KUKA KRL data list: Rack_Azul_Cerrar_D.dat

&ACCESS RVO1
&REL 85
&COMMENT CERRAR BANDEJAS PRG
&PARAM EDITMASK = *
&PARAM TEMPLATE = C:\KRC\Roboter\Template\vorgabe
&PARAM DISKPATH = KRC:\R1\Program\MAFELEC
DEFDAT  Rack_Azul_Cerrar_D
;FOLD EXTERNAL DECLARATIONS;%{PE}%MKUKATPBASIS,%CEXT,%VCOMMON,%P
;FOLD GRIPPERTECH EXT
EXT  H50 (INT  :IN,INT  :IN,INT  :IN,GRP_TYP  :IN )
;ENDFOLD (GRIPPERTECH EXT)
;FOLD SPOTTECH EXT
EXT  USERSPOT (S_COMMAND  :IN,SPOT_TYPE  :IN )
;ENDFOLD (SPOTTECH EXT)
;FOLD BASISTECH EXT;%{PE}%MKUKATPBASIS,%CEXT,%VEXT,%P
EXT  BAS (BAS_COMMAND  :IN,REAL  :IN )
DECL INT SUCCESS
;ENDFOLD (BASISTECH EXT)
;FOLD USER EXT;%{E}%MKUKATPUSER,%CEXT,%VEXT,%P
;Make your modifications here

;ENDFOLD (USER EXT)
;ENDFOLD (EXTERNAL DECLARATIONS)
DECL BASIS_SUGG_T LAST_BASIS={POINT1[] "P0                      ",POINT2[] "P0                      ",CP_PARAMS[] "CPDAT0                  ",PTP_PARAMS[] "PDAT0                   ",CONT[] "                        ",CP_VEL[] "1                       ",PTP_VEL[] "100                     ",SYNC_PARAMS[] "SYNCDAT                 ",SPL_NAME[] "S0                      ",A_PARAMS[] "ADAT0                   "}
DECL PDAT PH={VEL 100.000,ACC 100.000,APO_DIST 100.000,APO_MODE #CDIS,GEAR_JERK 50.0000,EXAX_IGN 0}
DECL E6POS XPOS_ESPERA_AREA1={X 112.943756,Y -227.851166,Z 2716.11304,A 36.2463837,B -15.5853510,C 56.0520973,S 3,T 42,E1 0.0,E2 0.0,E3 0.0,E4 0.0,E5 0.0,E6 0.0}
DECL FDAT FPOS_ESPERA_AREA1={TOOL_NO 9,BASE_NO 0,IPO_FRAME #BASE,POINT2[] " ",TQ_STATE FALSE}
DECL LDAT LL={VEL 2.00000,ACC 10.0000,APO_DIST 10.0000,APO_FAC 50.0000,AXIS_VEL 100.000,AXIS_ACC 100.000,ORI_TYP #VAR,CIRC_TYP #BASE,JERK_FAC 50.0000,GEAR_JERK 50.0000,EXAX_IGN 0}
DECL E6POS XPOS_AREA1_LIBRE={X -1304.04749,Y 95.8301,Z 2445.06763,A 84.0317841,B 0.238675669,C -89.1419449,S 6,T 59,E1 0.0,E2 0.0,E3 0.0,E4 0.0,E5 0.0,E6 0.0}
DECL FDAT FPOS_AREA1_LIBRE={TOOL_NO 9,BASE_NO 0,IPO_FRAME #BASE,POINT2[] " ",TQ_STATE FALSE}
DECL E6POS XP111={X 557.799622,Y -753.947571,Z -222.785736,A -88.9974060,B 13.7721291,C 89.1738281,S 6,T 58,E1 0.0,E2 0.0,E3 0.0,E4 0.0,E5 0.0,E6 0.0}
DECL FDAT FP111={TOOL_NO 1,BASE_NO 1,IPO_FRAME #BASE,POINT2[] " ",TQ_STATE FALSE}
DECL E6POS XP10={X 798.959167,Y -279.481934,Z 1381.33276,A 84.0317841,B 0.238675669,C -89.1419449,S 6,T 59,E1 0.0,E2 0.0,E3 0.0,E4 0.0,E5 0.0,E6 0.0}
DECL FDAT FP10={TOOL_NO 1,BASE_NO 2,IPO_FRAME #BASE,POINT2[] " ",TQ_STATE FALSE}
DECL E6POS XP110={X 704.303,Y -173.406952,Z -111.942,A 88.8908,B 0.942831039,C -90.1997757,S 2,T 43,E1 0.0,E2 0.0,E3 0.0,E4 0.0,E5 0.0,E6 0.0}
DECL FDAT FP110={TOOL_NO 2,BASE_NO 2,IPO_FRAME #BASE,POINT2[] " ",TQ_STATE FALSE}
DECL E6POS XP120={X 613.997192,Y -12.6072426,Z 50.9099464,A 86.9020615,B 2.85824347,C -89.1819077,S 2,T 43,E1 0.0,E2 0.0,E3 0.0,E4 0.0,E5 0.0,E6 0.0}
DECL FDAT FP120={TOOL_NO 2,BASE_NO 2,IPO_FRAME #BASE,POINT2[] " ",TQ_STATE FALSE}
DECL E6POS XP_ABRIR10={X -250.533554,Y -43.6507149,Z 2716.11304,A -84.6604385,B 6.50295877,C 57.2217522,S 3,T 42,E1 0.0,E2 0.0,E3 0.0,E4 0.0,E5 0.0,E6 0.0}
DECL FDAT FP_ABRIR10={TOOL_NO 9,BASE_NO 0,IPO_FRAME #BASE,POINT2[] " ",TQ_STATE FALSE}
DECL E6POS XP_AHOME={X -82.6595917,Y 188.465759,Z 3211.91699,A -95.2038803,B -13.5609741,C 10.5279636,S 2,T 43,E1 0.0,E2 0.0,E3 0.0,E4 0.0,E5 0.0,E6 0.0}
DECL FDAT FP_aHOME={TOOL_NO 9,BASE_NO 0,IPO_FRAME #BASE,POINT2[] " ",TQ_STATE FALSE}
DECL E6POS XIni_Cerrar_B1={X 596.412415,Y 736.011475,Z -172.103745,A 87.1854095,B 10.2055225,C -88.9196167,S 2,T 43,E1 0.0,E2 0.0,E3 0.0,E4 0.0,E5 0.0,E6 0.0}
DECL FDAT FIni_Cerrar_B1={TOOL_NO 2,BASE_NO 2,IPO_FRAME #BASE,POINT2[] " ",TQ_STATE FALSE}
DECL E6POS XAux_Cerrar_B1={X 588.737793,Y 569.274475,Z -354.425659,A 86.8103943,B 19.7198429,C -89.4653320,S 2,T 43,E1 0.0,E2 0.0,E3 0.0,E4 0.0,E5 0.0,E6 0.0}
DECL E6POS XFin_Cerrar_B1={X 586.341125,Y 418.554230,Z -648.000366,A 86.3078079,B 27.9656658,C -90.0449677,S 2,T 43,E1 0.0,E2 0.0,E3 0.0,E4 0.0,E5 0.0,E6 0.0}
DECL FDAT FFin_Cerrar_B1={TOOL_NO 2,BASE_NO 2,IPO_FRAME #BASE,POINT2[] "XAux_Cerrar_B1",TQ_STATE FALSE}
DECL E6POS XP0={X 632.645691,Y 303.475861,Z -186.174820,A -88.8950272,B 31.1322117,C 89.5053635,S 6,T 58,E1 0.0,E2 0.0,E3 0.0,E4 0.0,E5 0.0,E6 0.0}
DECL FDAT FP0={TOOL_NO 1,BASE_NO 1,IPO_FRAME #BASE,POINT2[] " ",TQ_STATE FALSE}
DECL E6POS XIni_Cerrar_B2={X 595.075134,Y 739.054,Z 45.4564934,A 87.7715607,B 2.41526031,C -90.0604706,S 2,T 43,E1 0.0,E2 0.0,E3 0.0,E4 0.0,E5 0.0,E6 0.0}
DECL FDAT FIni_Cerrar_B2={TOOL_NO 2,BASE_NO 2,IPO_FRAME #BASE,POINT2[] " ",TQ_STATE FALSE}
DECL E6POS XP1={X 633.606323,Y -740.251,Z -11.7250,A -89.0051498,B 9.17837143,C 89.0890656,S 6,T 58,E1 0.0,E2 0.0,E3 0.0,E4 0.0,E5 0.0,E6 0.0}
DECL FDAT FP1={TOOL_NO 1,BASE_NO 1,IPO_FRAME #BASE,POINT2[] " ",TQ_STATE FALSE}
DECL E6POS XAux_Cerrar_B2={X 587.798340,Y 417.710510,Z -431.910645,A 86.7692,B 24.2213230,C -90.6604462,S 2,T 43,E1 0.0,E2 0.0,E3 0.0,E4 0.0,E5 0.0,E6 0.0}
DECL E6POS XFin_Cerrar_B2={X 589.010254,Y 377.397522,Z -588.953735,A 86.3949585,B 28.6069508,C -90.8338776,S 2,T 43,E1 0.0,E2 0.0,E3 0.0,E4 0.0,E5 0.0,E6 0.0}
DECL FDAT FFin_Cerrar_B2={TOOL_NO 2,BASE_NO 2,IPO_FRAME #BASE,POINT2[] "XAux_Cerrar_B2",TQ_STATE FALSE}
DECL E6POS XP2={X 535.775818,Y 225.276917,Z -536.621948,A -91.0083771,B 14.9493265,C 94.2730637,S 6,T 58,E1 0.0,E2 0.0,E3 0.0,E4 0.0,E5 0.0,E6 0.0}
DECL FDAT FP2={TOOL_NO 1,BASE_NO 1,IPO_FRAME #BASE,POINT2[] " ",TQ_STATE FALSE}
DECL E6POS XP210={X 613.997192,Y -12.6072426,Z 50.9099464,A 86.9020615,B 2.85824347,C -89.1819077,S 2,T 43,E1 0.0,E2 0.0,E3 0.0,E4 0.0,E5 0.0,E6 0.0}
DECL FDAT FP210={TOOL_NO 2,BASE_NO 2,IPO_FRAME #BASE,POINT2[] " ",TQ_STATE FALSE}
DECL E6POS XP220={X 533.749146,Y -27.5535755,Z 294.696930,A 86.9283752,B 2.03337383,C -89.1903,S 2,T 43,E1 0.0,E2 0.0,E3 0.0,E4 0.0,E5 0.0,E6 0.0}
DECL FDAT FP220={TOOL_NO 2,BASE_NO 2,IPO_FRAME #BASE,POINT2[] " ",TQ_STATE FALSE}
DECL E6POS XP3={X 536.241516,Y 225.176605,Z 24.6719704,A -90.9851761,B 14.9447651,C 94.2668762,S 6,T 58,E1 0.0,E2 0.0,E3 0.0,E4 0.0,E5 0.0,E6 0.0}
DECL FDAT FP3={TOOL_NO 1,BASE_NO 1,IPO_FRAME #BASE,POINT2[] " ",TQ_STATE FALSE}
DECL E6POS XIni_Cerrar_B3={X 591.523193,Y 682.249634,Z 258.567474,A 86.9371643,B 3.42378807,C -89.3304749,S 2,T 43,E1 0.0,E2 0.0,E3 0.0,E4 0.0,E5 0.0,E6 0.0}
DECL FDAT FIni_Cerrar_B3={TOOL_NO 2,BASE_NO 2,IPO_FRAME #BASE,POINT2[] " ",TQ_STATE FALSE}
DECL E6POS XP4={X 633.606323,Y -740.251,Z -11.7250,A -89.0051498,B 9.17837143,C 89.0890656,S 6,T 58,E1 0.0,E2 0.0,E3 0.0,E4 0.0,E5 0.0,E6 0.0}
DECL FDAT FP4={TOOL_NO 1,BASE_NO 1,IPO_FRAME #BASE,POINT2[] " ",TQ_STATE FALSE}
DECL E6POS XAux_Cerrar_B3={X 594.214478,Y 611.080200,Z 74.3711472,A 86.8144608,B 12.5334587,C -90.4729614,S 2,T 43,E1 0.0,E2 0.0,E3 0.0,E4 0.0,E5 0.0,E6 0.0}
DECL E6POS XFin_Cerrar_B3={X 594.299866,Y 495.802765,Z -23.1475124,A 86.6915588,B 19.7912579,C -90.9023514,S 2,T 43,E1 0.0,E2 0.0,E3 0.0,E4 0.0,E5 0.0,E6 0.0}
DECL FDAT FFin_Cerrar_B3={TOOL_NO 2,BASE_NO 2,IPO_FRAME #BASE,POINT2[] "XAux_Cerrar_B3",TQ_STATE FALSE}
DECL E6POS XP5={X 535.775818,Y 225.276917,Z -194.099075,A -91.0083771,B 14.9493265,C 94.2730637,S 6,T 58,E1 0.0,E2 0.0,E3 0.0,E4 0.0,E5 0.0,E6 0.0}
DECL FDAT FP5={TOOL_NO 1,BASE_NO 1,IPO_FRAME #BASE,POINT2[] " ",TQ_STATE FALSE}
DECL E6POS XP310={X 533.749146,Y -27.5535755,Z 294.696930,A 86.9283752,B 2.03337383,C -89.1903,S 2,T 43,E1 0.0,E2 0.0,E3 0.0,E4 0.0,E5 0.0,E6 0.0}
DECL FDAT FP310={TOOL_NO 2,BASE_NO 2,IPO_FRAME #BASE,POINT2[] " ",TQ_STATE FALSE}
DECL E6POS XP320={X 530.175537,Y -40.1798019,Z 566.405701,A 86.9635239,B 0.231809333,C -89.0943146,S 2,T 43,E1 0.0,E2 0.0,E3 0.0,E4 0.0,E5 0.0,E6 0.0}
DECL FDAT FP320={TOOL_NO 2,BASE_NO 2,IPO_FRAME #BASE,POINT2[] " ",TQ_STATE FALSE}
DECL E6POS XP310_1={X 593.836731,Y 726.394348,Z 223.429489,A 86.8993149,B 3.44547296,C -89.9683228,S 2,T 43,E1 0.0,E2 0.0,E3 0.0,E4 0.0,E5 0.0,E6 0.0}
DECL FDAT FP310_1={TOOL_NO 2,BASE_NO 2,IPO_FRAME #BASE,POINT2[] " ",TQ_STATE FALSE}
DECL E6POS XP6={X 536.241516,Y 225.176605,Z 24.6719704,A -90.9851761,B 14.9447651,C 94.2668762,S 6,T 58,E1 0.0,E2 0.0,E3 0.0,E4 0.0,E5 0.0,E6 0.0}
DECL FDAT FP6={TOOL_NO 1,BASE_NO 1,IPO_FRAME #BASE,POINT2[] " ",TQ_STATE FALSE}
DECL E6POS XIni_Cerrar_B4={X 582.265930,Y 720.715637,Z 474.957,A 86.9055099,B 6.88711309,C -89.5095520,S 2,T 43,E1 0.0,E2 0.0,E3 0.0,E4 0.0,E5 0.0,E6 0.0}
DECL FDAT FIni_Cerrar_B4={TOOL_NO 2,BASE_NO 2,IPO_FRAME #BASE,POINT2[] " ",TQ_STATE FALSE}
DECL E6POS XP7={X 633.606323,Y -740.251,Z -11.7250,A -89.0051498,B 9.17837143,C 89.0890656,S 6,T 58,E1 0.0,E2 0.0,E3 0.0,E4 0.0,E5 0.0,E6 0.0}
DECL FDAT FP7={TOOL_NO 1,BASE_NO 1,IPO_FRAME #BASE,POINT2[] " ",TQ_STATE FALSE}
DECL E6POS XAux_Cerrar_B4={X 576.527588,Y 424.657928,Z -21.2641106,A 87.9251328,B 24.5308399,C -90.4093552,S 2,T 43,E1 0.0,E2 0.0,E3 0.0,E4 0.0,E5 0.0,E6 0.0}
DECL E6POS XFin_Cerrar_B4={X 576.502,Y 330.746521,Z -306.611084,A 88.2723389,B 22.7116070,C -90.3397293,S 2,T 43,E1 0.0,E2 0.0,E3 0.0,E4 0.0,E5 0.0,E6 0.0}
DECL FDAT FFin_Cerrar_B4={TOOL_NO 2,BASE_NO 2,IPO_FRAME #BASE,POINT2[] "XAux_Cerrar_B4",TQ_STATE FALSE}
DECL E6POS XP8={X 535.775818,Y 225.276917,Z -194.099075,A -91.0083771,B 14.9493265,C 94.2730637,S 6,T 58,E1 0.0,E2 0.0,E3 0.0,E4 0.0,E5 0.0,E6 0.0}
DECL FDAT FP8={TOOL_NO 1,BASE_NO 1,IPO_FRAME #BASE,POINT2[] " ",TQ_STATE FALSE}
DECL E6POS XP410={X 530.175537,Y -40.1798019,Z 566.405701,A 86.9635239,B 0.231809333,C -89.0943146,S 2,T 43,E1 0.0,E2 0.0,E3 0.0,E4 0.0,E5 0.0,E6 0.0}
DECL FDAT FP410={TOOL_NO 2,BASE_NO 2,IPO_FRAME #BASE,POINT2[] " ",TQ_STATE FALSE}
DECL E6POS XP410_1={X 583.801,Y 728.139099,Z 438.754639,A 86.9037552,B 7.08309031,C -89.5218811,S 2,T 43,E1 0.0,E2 0.0,E3 0.0,E4 0.0,E5 0.0,E6 0.0}
DECL FDAT FP410_1={TOOL_NO 2,BASE_NO 2,IPO_FRAME #BASE,POINT2[] " ",TQ_STATE FALSE}
DECL E6POS XP420={X 796.310425,Y -36.4565620,Z 1201.42468,A 84.0344,B 0.236838102,C -89.1263580,S 6,T 59,E1 0.0,E2 0.0,E3 0.0,E4 0.0,E5 0.0,E6 0.0}
DECL FDAT FP420={TOOL_NO 2,BASE_NO 2,IPO_FRAME #BASE,POINT2[] " ",TQ_STATE FALSE}
DECL E6POS XP9={X 536.241516,Y 225.176605,Z 24.6719704,A -90.9851761,B 14.9447651,C 94.2668762,S 6,T 58,E1 0.0,E2 0.0,E3 0.0,E4 0.0,E5 0.0,E6 0.0}
DECL FDAT FP9={TOOL_NO 1,BASE_NO 1,IPO_FRAME #BASE,POINT2[] " ",TQ_STATE FALSE}
DECL E6POS XIni_Cerrar_B5={X 547.158386,Y 717.412231,Z 958.713684,A 91.7971573,B 9.40811539,C -90.5130844,S 6,T 59,E1 0.0,E2 0.0,E3 0.0,E4 0.0,E5 0.0,E6 0.0}
DECL FDAT FIni_Cerrar_B5={TOOL_NO 2,BASE_NO 2,IPO_FRAME #BASE,POINT2[] " ",TQ_STATE FALSE}
DECL E6POS XP11={X 633.606323,Y -740.251,Z -11.7250,A -89.0051498,B 9.17837143,C 89.0890656,S 6,T 58,E1 0.0,E2 0.0,E3 0.0,E4 0.0,E5 0.0,E6 0.0}
DECL FDAT FP11={TOOL_NO 1,BASE_NO 1,IPO_FRAME #BASE,POINT2[] " ",TQ_STATE FALSE}
DECL E6POS XAux_Cerrar_B5={X 558.484192,Y 280.618256,Z 418.164581,A 92.4280930,B 33.5212364,C -88.3598862,S 6,T 59,E1 0.0,E2 0.0,E3 0.0,E4 0.0,E5 0.0,E6 0.0}
DECL E6POS XFin_Cerrar_B5={X 548.725647,Y 142.679794,Z -91.2902527,A 93.2127762,B 51.9579430,C -86.3543167,S 6,T 59,E1 0.0,E2 0.0,E3 0.0,E4 0.0,E5 0.0,E6 0.0}
DECL FDAT FFin_Cerrar_B5={TOOL_NO 2,BASE_NO 2,IPO_FRAME #BASE,POINT2[] "XAux_Cerrar_B5",TQ_STATE FALSE}
DECL E6POS XP12={X 535.775818,Y 225.276917,Z -194.099075,A -91.0083771,B 14.9493265,C 94.2730637,S 6,T 58,E1 0.0,E2 0.0,E3 0.0,E4 0.0,E5 0.0,E6 0.0}
DECL FDAT FP12={TOOL_NO 1,BASE_NO 1,IPO_FRAME #BASE,POINT2[] " ",TQ_STATE FALSE}
DECL E6POS XP510={X 796.310425,Y -36.4565620,Z 1201.42468,A 84.0344,B 0.236838102,C -89.1263580,S 6,T 59,E1 0.0,E2 0.0,E3 0.0,E4 0.0,E5 0.0,E6 0.0}
DECL FDAT FP510={TOOL_NO 2,BASE_NO 2,IPO_FRAME #BASE,POINT2[] " ",TQ_STATE FALSE}
DECL E6POS XP510_1={X 560.767,Y 703.689941,Z 903.786133,A 91.7950592,B 9.40895271,C -90.5137787,S 6,T 59,E1 0.0,E2 0.0,E3 0.0,E4 0.0,E5 0.0,E6 0.0}
DECL FDAT FP510_1={TOOL_NO 2,BASE_NO 2,IPO_FRAME #BASE,POINT2[] " ",TQ_STATE FALSE}
DECL E6POS XP520={X 796.200256,Y -279.947296,Z 1201.35449,A 84.0317841,B 0.238675669,C -89.1419449,S 6,T 59,E1 0.0,E2 0.0,E3 0.0,E4 0.0,E5 0.0,E6 0.0}
DECL FDAT FP520={TOOL_NO 2,BASE_NO 2,IPO_FRAME #BASE,POINT2[] " ",TQ_STATE FALSE}
DECL E6POS XP210_1={X 594.377869,Y 711.943726,Z 1.48922753,A 87.8185272,B 10.3139572,C -90.3250122,S 2,T 43,E1 0.0,E2 0.0,E3 0.0,E4 0.0,E5 0.0,E6 0.0}
DECL FDAT FP210_1={TOOL_NO 2,BASE_NO 2,IPO_FRAME #BASE,POINT2[] " ",TQ_STATE FALSE}
DECL E6POS XP110_1={X 591.121521,Y 739.826843,Z -203.536621,A 87.1612778,B 12.3881922,C -89.0297928,S 2,T 43,E1 0.0,E2 0.0,E3 0.0,E4 0.0,E5 0.0,E6 0.0}
DECL FDAT FP110_1={TOOL_NO 2,BASE_NO 2,IPO_FRAME #BASE,POINT2[] " ",TQ_STATE FALSE}
DECL E6POS XP_FIN={X 798.959167,Y 2019.51807,Z 1386.33276,A 84.0317841,B 0.238675669,C -89.1419449,S 6,T 59,E1 0.0,E2 0.0,E3 0.0,E4 0.0,E5 0.0,E6 0.0}
DECL FDAT FP_FIN={TOOL_NO 1,BASE_NO 1,IPO_FRAME #BASE,POINT2[] " ",TQ_STATE FALSE}
DECL E6POS XPCONEX={X 850.773865,Y 724.424316,Z 273.456970,A -87.1000290,B -0.167936072,C 179.536102,S 2,T 42,E1 0.0,E2 0.0,E3 0.0,E4 0.0,E5 0.0,E6 0.0}
DECL FDAT FPCONEX={TOOL_NO 9,BASE_NO 1,IPO_FRAME #BASE,POINT2[] " ",TQ_STATE FALSE}
DECL PDAT PPDAT1={VEL 100.000,ACC 100.000,APO_DIST 100.000,GEAR_JERK 50.0000,EXAX_IGN 0}
DECL E6POS XP13={X 576.700562,Y 552.299805,Z 243.688065,A 87.4606,B 16.4706306,C -90.0445557,S 2,T 43,E1 0.0,E2 0.0,E3 0.0,E4 0.0,E5 0.0,E6 0.0}
DECL E6POS XP14={X 578.304749,Y 463.264435,Z 80.0048523,A 87.7890167,B 25.2298965,C -90.4399,S 2,T 43,E1 0.0,E2 0.0,E3 0.0,E4 0.0,E5 0.0,E6 0.0}
DECL FDAT FP14={TOOL_NO 2,BASE_NO 2,IPO_FRAME #BASE,POINT2[] "XP13",TQ_STATE FALSE}
DECL LDAT LM={VEL 2.00000,ACC 50.0000,APO_DIST 25.0000,APO_FAC 50.0000,AXIS_VEL 100.000,AXIS_ACC 100.000,ORI_TYP #VAR,CIRC_TYP #BASE,JERK_FAC 50.0000,GEAR_JERK 50.0000,EXAX_IGN 0}
DECL E6POS XP15={X 582.600769,Y 398.596130,Z -683.197,A 88.2728806,B 32.2285957,C -90.3512115,S 2,T 43,E1 0.0,E2 0.0,E3 0.0,E4 0.0,E5 0.0,E6 0.0}
DECL E6POS XP16={X 582.300232,Y 347.256104,Z -927.256226,A 88.2825623,B 32.2318840,C -90.3522,S 2,T 43,E1 0.0,E2 0.0,E3 0.0,E4 0.0,E5 0.0,E6 0.0}
DECL FDAT FP16={TOOL_NO 2,BASE_NO 2,IPO_FRAME #BASE,POINT2[] "XP15",TQ_STATE FALSE}
DECL E6POS XP17={X 592.372498,Y 363.706818,Z -726.446899,A 86.4632416,B 26.5387630,C -90.6878281,S 2,T 43,E1 0.0,E2 0.0,E3 0.0,E4 0.0,E5 0.0,E6 0.0}
DECL FDAT FP17={TOOL_NO 2,BASE_NO 2,IPO_FRAME #BASE,POINT2[] " ",TQ_STATE FALSE}
DECL E6POS XP18={X 590.012146,Y 356.174652,Z -511.359863,A 87.8676529,B 17.3292198,C -90.2225876,S 2,T 43,E1 0.0,E2 0.0,E3 0.0,E4 0.0,E5 0.0,E6 0.0}
DECL FDAT FP18={TOOL_NO 2,BASE_NO 2,IPO_FRAME #BASE,POINT2[] " ",TQ_STATE FALSE}
DECL PDAT PM={VEL 100.000,ACC 50.0000,APO_DIST 100.000,APO_MODE #CDIS,GEAR_JERK 50.0000,EXAX_IGN 0}
DECL E6POS XP01={X 1263.42725,Y 22.2543468,Z 976.105774,A 86.6829224,B -17.0911541,C -157.124573,S 2,T 35,E1 0.0,E2 0.0,E3 0.0,E4 0.0,E5 0.0,E6 0.0}
DECL FDAT FP01={TOOL_NO 1,BASE_NO 2,IPO_FRAME #BASE,POINT2[] " ",TQ_STATE FALSE}
DECL E6POS XP19={X 557.763123,Y 1999.29968,Z 884.990723,A 113.755737,B -9.84294605,C -110.000359,S 2,T 43,E1 0.0,E2 0.0,E3 0.0,E4 0.0,E5 0.0,E6 0.0}
DECL FDAT FP19={TOOL_NO 1,BASE_NO 1,IPO_FRAME #BASE,POINT2[] " ",TQ_STATE FALSE}
DECL PDAT PPDAT2={VEL 100.000,ACC 100.000,APO_DIST 100.000,APO_MODE #CDIS,GEAR_JERK 50.0000,EXAX_IGN 0}
DECL LDAT LCPDAT1={VEL 2.00000,ACC 25.0000,APO_DIST 100.000,APO_FAC 50.0000,AXIS_VEL 100.000,AXIS_ACC 100.000,ORI_TYP #VAR,CIRC_TYP #BASE,JERK_FAC 50.0000,GEAR_JERK 50.0000,EXAX_IGN 0}
DECL E6POS XP20={X 547.583,Y 152.647522,Z -98.5626907,A 92.8167801,B 46.3733635,C -86.8326721,S 6,T 59,E1 0.0,E2 0.0,E3 0.0,E4 0.0,E5 0.0,E6 0.0}
DECL FDAT FP20={TOOL_NO 2,BASE_NO 2,IPO_FRAME #BASE,POINT2[] " ",TQ_STATE FALSE}
ENDDAT
